// TIA Portal V18 export
// export: Created 2023-08-15T13:42:57.7282388Z, ExportSetting WithDefaults, DisplayName Totally Integrated Automation Portal, DisplayVersion V18 Update 2, DisplayName TIA Portal Openness, DisplayVersion V18 Update 2, DisplayName TIA Portal Version Control Interface, DisplayVersion V18, DisplayName SINAMICS Startdrive Advanced, DisplayVersion V18, DisplayName SINAMICS Startdrive G130, G150, S120, S150, SINAMICS MV, S210, DisplayVersion V18, DisplayName SINAMICS Startdrive G110M, G120, G120C, G120D, G120P, G115D, DisplayVersion V18, DisplayName STEP 7 Professional, DisplayVersion V18 Update 2, DisplayName STEP 7 Safety, DisplayVersion V18, DisplayName WinCC Advanced / Unified PC, DisplayVersion V18 Update 2
DATA_BLOCK "SinaSpeed2_DB"   // DB1
VERSION : 0.1
// stored: AutoNumber true, DBAccessibleFromOPCUA true, DBAccessibleFromWebserver true, InstanceOfName SinaSpeed2, InstanceOfType FB
"SinaSpeed2"
   // VAR_INPUT
   //    EnableAxis : Bool;
   //    AckError : Bool;
   //    SpeedSp : Real;
   //    RefSpeed : Real;
   //    ConfigAxis : Word;
   //    HWIDSTW : HW_IO;
   //    HWIDZSW : HW_IO;
   //    Input_1 : Int;
   // END_VAR
   // VAR_OUTPUT
   //    AxisEnabled : Bool;
   //    Lockout : Bool;
   //    ActVelocity : Real;
   //    Error : Bool;
   //    Status : Word;
   //    DiagId : Word;
   // END_VAR
   // VAR
   //    STW1 : Word;
   //    VelocitySP : Word;
   //    ZSW1 : Word;
   //    VelocityAV : Word;
   //    testarvo : Word;
   // END_VAR
BEGIN
END_DATA_BLOCK
